Staubli VAL3: MoveId.dtx

mdesc mNomSpeed
jointRx jJ
mdesc mMdesc
tool tTool = {fatherId=flange[0], ioLink=valve1}
